FUNCTION_BLOCK Analogue
VAR_INPUT
	Value:REAL;
	Raw_min:REAL;
	Raw_max:REAL;
	Scaled_min:REAL;
	Scaled_max:REAL;
	HH_setpoint:REAL := 1.000000E+008; (*The default value prevents the output from triggering if no setpoint is given*)
	H_setpoint:REAL := 1.000000E+008;
	L_setpoint:REAL := -1.000000E+008;
	ll_setpoint:REAL := -1.000000E+008;
	Hysteresis:REAL;
	Filter_time:TIME;
	Alarm_inhibit_time:TIME;
	HMI_min:REAL;
	HMI_max:REAL;
	Colour_scheme:INT;
END_VAR
VAR_OUTPUT
	Scaled_value:REAL;
	HH:BOOL;
	H:BOOL;
	L:BOOL;
	LL:BOOL;
	HMI:dut_hmi_Analogue;
END_VAR
VAR
	FB_CTRL_LEAD_LAG_0: FB_CTRL_LEAD_LAG;
	Lead_lag_params:ST_CTRL_LEAD_LAG_PARAMS;
	Hys_params:ST_CTRL_HYSTERESIS_PARAMS;
	FB_CTRL_HYSTERESIS_0: FB_CTRL_HYSTERESIS;
	TON_0: TON;
	FB_CTRL_HYSTERESIS_1: FB_CTRL_HYSTERESIS;
	TON_1: TON;
	FB_CTRL_HYSTERESIS_2: FB_CTRL_HYSTERESIS;
	TON_2: TON;
	FB_CTRL_HYSTERESIS_3: FB_CTRL_HYSTERESIS;
	TON_3: TON;
END_VAR

Analogue_m();
Analogue_HMI();

METHOD Analogue_HMI
VAR_INPUT
END_VAR
VAR_INST // added by the converter: edge detectors and wires of the graphical bodies
    _w1, _w2, _w3, _w4, _w5, _w6, _w7 : ANY;
END_VAR
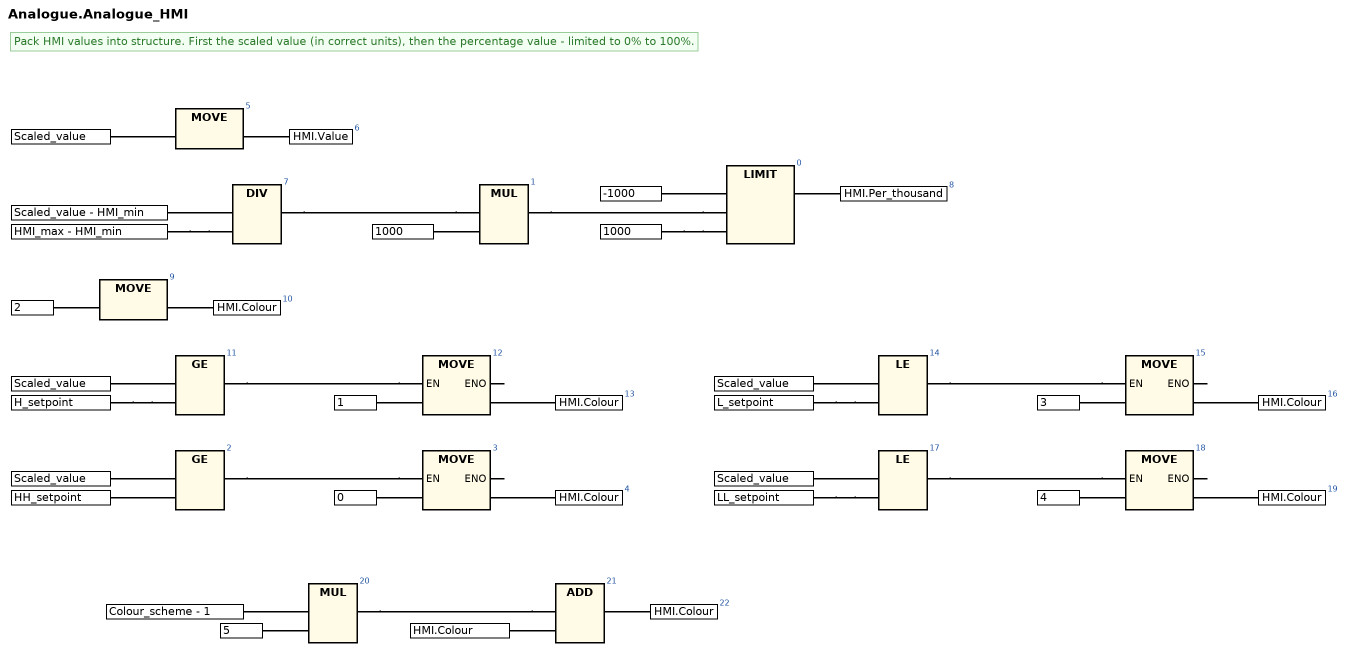
_w2 := LIMIT(-1000, _w1, 1000);
_w1 := _w3 * 1000;
IF Scaled_value >= HH_setpoint THEN _w4 := 0; END_IF
HMI.Colour := _w4;
// Pack HMI values into structure. First the scaled value (in correct units), then the percentage value - limited to 0% to 100%.
HMI.Value := Scaled_value;
_w3 := (Scaled_value - HMI_min) / (HMI_max - HMI_min);
HMI.Per_thousand := _w2;
HMI.Colour := 2;
IF Scaled_value >= H_setpoint THEN _w5 := 1; END_IF
HMI.Colour := _w5;
IF Scaled_value <= L_setpoint THEN _w6 := 3; END_IF
HMI.Colour := _w6;
IF Scaled_value <= LL_setpoint THEN _w7 := 4; END_IF
HMI.Colour := _w7;
HMI.Colour := (Colour_scheme - 1) * 5 + HMI.Colour;
END_METHOD

METHOD Analogue_m
VAR_INPUT
END_VAR
{warning "TODO: the LEAD LAG filter needs to be looked at by Bret so that he can make sure it does what he needs it to."}
{warning "TODO: the HYST FB needs to be looked at by Bret so that he can make sure it does what he needs it to."}
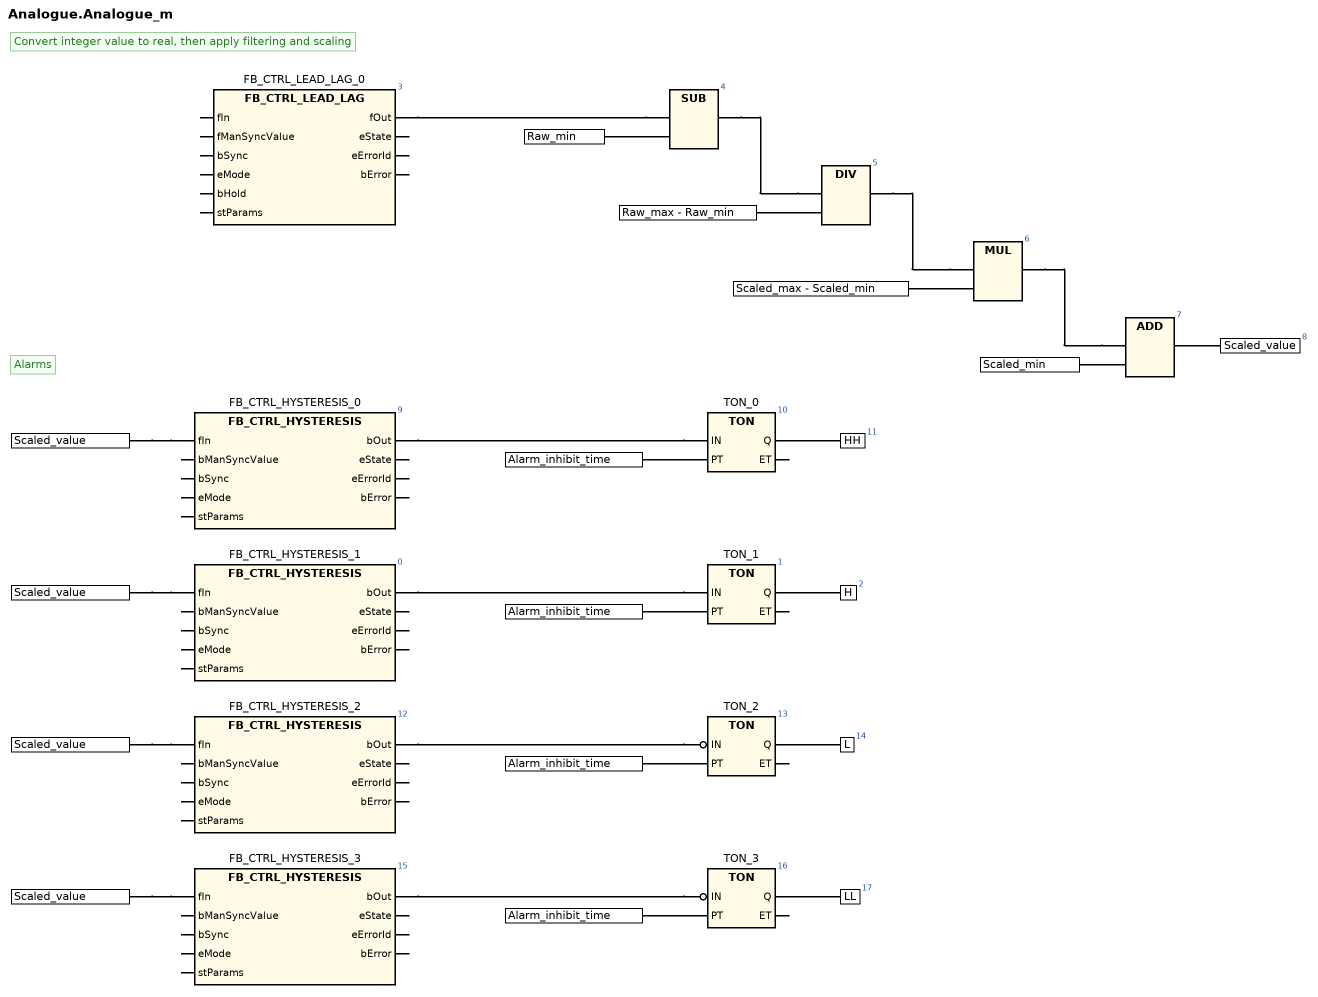
FB_CTRL_HYSTERESIS_1(fIn := Scaled_value); // FB_CTRL_HYSTERESIS
TON_1(IN := FB_CTRL_HYSTERESIS_1.bOut, PT := Alarm_inhibit_time); // TON
H := TON_1.Q;
// Convert integer value to real, then apply filtering and scaling
FB_CTRL_LEAD_LAG_0(); // FB_CTRL_LEAD_LAG
Scaled_value := ((FB_CTRL_LEAD_LAG_0.fOut - Raw_min) / (Raw_max - Raw_min)) * (Scaled_max - Scaled_min) + Scaled_min;
// Alarms
FB_CTRL_HYSTERESIS_0(fIn := Scaled_value); // FB_CTRL_HYSTERESIS
TON_0(IN := FB_CTRL_HYSTERESIS_0.bOut, PT := Alarm_inhibit_time); // TON
HH := TON_0.Q;
FB_CTRL_HYSTERESIS_2(fIn := Scaled_value); // FB_CTRL_HYSTERESIS
TON_2(IN := NOT FB_CTRL_HYSTERESIS_2.bOut, PT := Alarm_inhibit_time); // TON
L := TON_2.Q;
FB_CTRL_HYSTERESIS_3(fIn := Scaled_value); // FB_CTRL_HYSTERESIS
TON_3(IN := NOT FB_CTRL_HYSTERESIS_3.bOut, PT := Alarm_inhibit_time); // TON
LL := TON_3.Q;
END_METHOD

END_FUNCTION_BLOCK

(* stored: Version 1.1.0.1, ProductVersion 3.1.4024.0
   POU Analogue: Id {7994f1f8-4814-4f45-8931-1ef83acd9447}, SpecialFunc None
   Method Analogue_HMI: Id {19ea1c72-a486-4826-9aea-6b6a476be412}
   Method Analogue_m: Id {1e5fdfaf-114c-45d0-84d8-15f2bb60051a} *)
